FUNCTION_BLOCK FB_CargarBase_SFC
VAR_INPUT
    // SFC-Flags
    SFCPause: BOOL;
    SFCReset: BOOL;
    
    // Indicadores de sincronizacion
    Ack: BOOL := TRUE;
    Execute: BOOL;
    
    // Entradas
    ManipuladorDetras: BOOL; // Sobre el pale
    ManipuladorMedio: BOOL := TRUE; // En la vertical
    ManipuladorDelante: BOOL; // Sobre el punto de trasvase de la presa\
    ManipuladorVacioObtenido: BOOL;
END_VAR
VAR_OUTPUT
    // Indicadores de sincronizacion
    Done: BOOL;
    Ready: BOOL;

    // Salidas
    ManipuladorAdelante: BOOL; // Hacia el punto de trasvase de la prensa
    ManipuladorAtras: BOOL; // Hacia el pale
    ManipuladorSucciona: BOOL;
END_VAR
VAR
END_VAR

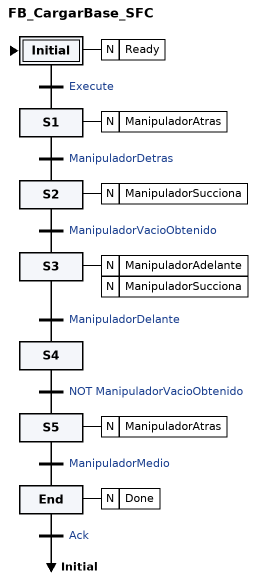
INITIAL_STEP Initial:
    Ready(N);
END_STEP
TRANSITION FROM Initial TO S1
    := Execute;
END_TRANSITION
STEP S1:
    ManipuladorAtras(N);
END_STEP
TRANSITION FROM S1 TO S2
    := ManipuladorDetras;
END_TRANSITION
STEP S2:
    ManipuladorSucciona(N);
END_STEP
TRANSITION FROM S2 TO S3
    := ManipuladorVacioObtenido;
END_TRANSITION
STEP S3:
    ManipuladorAdelante(N);
    ManipuladorSucciona(N);
END_STEP
TRANSITION FROM S3 TO S4
    := ManipuladorDelante;
END_TRANSITION
STEP S4:
END_STEP
TRANSITION FROM S4 TO S5
    := NOT ManipuladorVacioObtenido;
END_TRANSITION
STEP S5:
    ManipuladorAtras(N);
END_STEP
TRANSITION FROM S5 TO End
    := ManipuladorMedio;
END_TRANSITION
STEP End:
    Done(N);
END_STEP
TRANSITION FROM End TO Initial
    := Ack;
END_TRANSITION

END_FUNCTION_BLOCK

(* stored: Version 1.1.0.1, ProductVersion 3.1.4024.12
   POU FB_CargarBase_SFC: Id {1da4f34f-7783-47c8-bdf4-e619b098379a}, SpecialFunc None *)
